FUNCTION_BLOCK GRIPPER_GIMATIC EXTENDS FB_1_Tool
VAR_INPUT
	    
    pUR : POINTER TO ROBOT_UR; // UR instance that physically carries this gripper.
    nToolOutput : USINT := 0; // Tool output used by the Gimatic interface.
    bGripLevel : BOOL := TRUE; // Electrical level that means "grip".
END_VAR
VAR_OUTPUT
    bConfigured : BOOL;
    bGripCmd     : BOOL;
END_VAR

VAR
    _nConfigState : USINT := 0;
END_VAR

METHOD Grip : eResult
VAR_INPUT
END_VAR
IF bGripLevel THEN
	Grip := SetGripperOutput(TRUE);
ELSE
	Grip := SetGripperOutput(FALSE);
END_IF
END_METHOD

METHOD PROTECTED onActivate : eResult
VAR_INPUT
END_VAR

VAR
	eParentResult: eResult;
	myResult: ERESULT;
END_VAR

VAR //YOUR CODE
	succ : BOOL;
END_VAR
eParentResult := SUPER^.onActivate();
myResult := NONE;

IF (pUR = 0) OR NOT bConfigured THEN
    Messenger.AddWarn(eMessageCategories.StateMachine, Path,
        'Gimatic gripper cannot activate because it is not configured');
    myResult := FAILURE;
ELSE
    myResult := SUCCESS;
END_IF

onActivate := CombineResults(eParentResult, myResult);
END_METHOD

METHOD PROTECTED onCleanup : eResult
VAR_INPUT
END_VAR

VAR
	eParentResult: eResult;
	myResult: ERESULT;
END_VAR

VAR //YOUR CODE
	succ : BOOL;
END_VAR
eParentResult := SUPER^.onCleanup();
bConfigured := FALSE;
bGripCmd := FALSE;
_nConfigState := 0;
myResult := SUCCESS;
onCleanup := CombineResults(eParentResult, myResult);
END_METHOD

METHOD PROTECTED onConfigure : eResult
VAR_INPUT
END_VAR

VAR
	eParentResult: eResult;
	myResult: ERESULT;
END_VAR

VAR //YOUR CODE
	succ : BOOL;
END_VAR
eParentResult := SUPER^.onConfigure();

//--------------------------------------------------
myResult := NONE;
//--------------------------------------------------

IF pUR = 0 THEN

    SetRecoveryMode(Mode := eRecoveryMode.ManualActionRequired);
    Messenger.AddError(
        eMessageCategories.Undefined,
        Name,
        'Gimatic gripper: pUR is not assigned'
    );

    bConfigured := FALSE;
    _nConfigState := 0;
    myResult := ERROR;

ELSIF nToolOutput > 1 THEN

    SetRecoveryMode(Mode := eRecoveryMode.ManualActionRequired);
    Messenger.AddError(
        eMessageCategories.Undefined,
        Name,
        'Gimatic gripper: nToolOutput must be 0 or 1'
    );

    bConfigured := FALSE;
    _nConfigState := 0;
    myResult := ERROR;

ELSIF pUR^.UR_COMM.Script.bError THEN

    SetRecoveryMode(Mode := eRecoveryMode.Automatic);
    Messenger.AddError(
        eMessageCategories.HardwareFailure,
        Name,
        'Gimatic gripper: URScript interface error'
    );

    bConfigured := FALSE;
    _nConfigState := 0;
    myResult := ERROR;

ELSE

    CASE _nConfigState OF

        0:
            bConfigured := FALSE;

            // Wait until URScript interface is available.
            IF pUR^.UR_COMM.Script.bOperational THEN

                succ :=
                    pUR^.UR_COMM.Script.ClearScript()
                    AND pUR^.UR_COMM.Script.AppendLine(
                        sLine := 'def plc_gripper_config():'
                    )
                    AND pUR^.UR_COMM.Script.AppendLine(
                        sLine := '  set_tool_voltage(24)'
                    );

                IF succ THEN

                    IF nToolOutput = 0 THEN

                        succ :=
                            pUR^.UR_COMM.Script.AppendLine(
                                sLine := '  set_tool_digital_output_mode(0,1)'
                            );

                    ELSE

                        succ :=
                            pUR^.UR_COMM.Script.AppendLine(
                                sLine := '  set_tool_digital_output_mode(1,1)'
                            );

                    END_IF

                END_IF

                succ := succ
                    AND pUR^.UR_COMM.Script.AppendLine(
                        sLine := 'end'
                    )
                    AND pUR^.UR_COMM.Script.SendBuffered();

                IF succ THEN
                    _nConfigState := 10;
                END_IF

            END_IF


        10:
            // Wait until the script FB starts sending.
            IF pUR^.UR_COMM.Script.bScriptSent THEN

                bConfigured := TRUE;
                _nConfigState := 100;

            ELSIF pUR^.UR_COMM.Script.bBusy THEN

                _nConfigState := 20;

            END_IF


        20:
            // Wait until sending is finished.
            IF pUR^.UR_COMM.Script.bError THEN
                SetRecoveryMode(Mode := eRecoveryMode.Automatic);
                Messenger.AddError(eMessageCategories.HardwareFailure, Name,
                    'Gimatic gripper: URScript interface error');

                _nConfigState := 0;
                bConfigured := FALSE;
                myResult := ERROR;

            ELSIF
                pUR^.UR_COMM.Script.bScriptSent
                OR NOT pUR^.UR_COMM.Script.bBusy
            THEN

                bConfigured := TRUE;
                _nConfigState := 100;

            END_IF


        100:
            bConfigured := TRUE;

            myResult := SUCCESS;

    END_CASE

END_IF

//--------------------------------------------------

onConfigure := CombineResults(
    eParentResult,
    myResult
);
END_METHOD

METHOD PROTECTED onDeactivate : eResult
VAR_INPUT
END_VAR

VAR
	eParentResult: eResult;
	myResult: ERESULT;
END_VAR

VAR //YOUR CODE
	succ : BOOL;
END_VAR
eParentResult := SUPER^.onDeactivate();
//--------------------------------------------------
myResult:=NONE;
// ----- YOUR CODE HERE (incl. Alarms) -------------

myResult:=SUCCESS;

// ----- END YOUR CODE -----------------------------
//--------------------------------------------------
onDeactivate := CombineResults(eParentResult,myResult);
END_METHOD

METHOD PROTECTED onError : eResult
VAR_INPUT
END_VAR

VAR
	eParentResult: eResult;
	myResult: ERESULT;
END_VAR

VAR //YOUR CODE
	succ : BOOL;
END_VAR
eParentResult := SUPER^.onError();
myResult := NONE;

bConfigured := FALSE;
_nConfigState := 0;

IF (pUR = 0) OR (nToolOutput > 1) THEN
    SetRecoveryMode(Mode := eRecoveryMode.ManualActionRequired);
    RequireNewAcknowledgement();
ELSIF pUR^.UR_COMM.State = eState.ErrorProcessing THEN
    SetRecoveryMode(Mode := pUR^.UR_COMM.RecoveryMode);
ELSIF pUR^.UR_COMM.Script.bBusy OR pUR^.UR_COMM.Script.bError THEN
    myResult := NONE;
ELSE
    myResult := SUCCESS;
END_IF

onError := CombineResults(eParentResult, myResult);
END_METHOD

METHOD PROTECTED onShutdown : eResult
VAR_INPUT
END_VAR

VAR
	eParentResult: eResult;
	myResult: ERESULT;
END_VAR

VAR //YOUR CODE
	succ : BOOL;
END_VAR
eParentResult := SUPER^.onShutdown();
//--------------------------------------------------
myResult:=NONE;
// ----- YOUR CODE HERE (incl. Alarms) -------------

// Do not release automatically on shutdown.
bConfigured := FALSE;
_nConfigState := 0;

myResult:=SUCCESS;


// ----- END YOUR CODE -----------------------------
//--------------------------------------------------
onShutdown := CombineResults(eParentResult,myResult);
END_METHOD

METHOD Release : eResult
VAR_INPUT
END_VAR
IF bGripLevel THEN
	Release := SetGripperOutput(FALSE);
ELSE
	Release := SetGripperOutput(TRUE);
END_IF
END_METHOD

METHOD SetGripperOutput : eResult
VAR_INPUT
	bValue: BOOL;
END_VAR
VAR
    succ : BOOL;
END_VAR

SetGripperOutput := NONE;

IF pUR = 0 THEN
    SetRecoveryMode(Mode := eRecoveryMode.ManualActionRequired);
    SetGripperOutput := ERROR;
	Messenger.AddError(eMessageCategories.MissingData,Path,'pUR is 0');
    RETURN;
END_IF

IF NOT bConfigured THEN
    SetRecoveryMode(Mode := eRecoveryMode.AcknowledgeRequired);
    SetGripperOutput := ERROR;
	Messenger.AddError(eMessageCategories.StateMachine,Path,'Gripper is not configured: OnConfigure');
    RETURN;
END_IF

IF pUR^.UR_COMM.Script.bError THEN
    SetRecoveryMode(Mode := eRecoveryMode.AcknowledgeRequired);
    SetGripperOutput := ERROR;
	Messenger.AddError(eMessageCategories.Undefined,Path,'UR_COMM is in Error');
    RETURN;
END_IF

// Do not overwrite a URScript command that is already being transmitted.
IF pUR^.UR_COMM.Script.bBusy THEN
    RETURN;
END_IF

IF NOT pUR^.UR_COMM.Script.ClearScript() THEN
    RETURN;
END_IF

IF NOT pUR^.UR_COMM.Script.AppendLine(
    sLine := 'def plc_grip():'
) THEN
    SetGripperOutput := ERROR;
    RETURN;
END_IF

IF nToolOutput = 0 THEN

    IF bValue THEN
        succ := pUR^.UR_COMM.Script.AppendLine(
            sLine := '  set_tool_digital_out(0,True)'
        );
    ELSE
        succ := pUR^.UR_COMM.Script.AppendLine(
            sLine := '  set_tool_digital_out(0,False)'
        );
    END_IF

ELSIF nToolOutput = 1 THEN

    IF bValue THEN
        succ := pUR^.UR_COMM.Script.AppendLine(
            sLine := '  set_tool_digital_out(1,True)'
        );
    ELSE
        succ := pUR^.UR_COMM.Script.AppendLine(
            sLine := '  set_tool_digital_out(1,False)'
        );
    END_IF

ELSE
    SetRecoveryMode(Mode := eRecoveryMode.ManualActionRequired);
    SetGripperOutput := ERROR;
    Messenger.AddError(eMessageCategories.StateMachine, Path, 'Invalid Gimatic tool output');
    RETURN;
END_IF

succ := succ
    AND pUR^.UR_COMM.Script.AppendLine(
        sLine := 'end'
    )
    AND pUR^.UR_COMM.Script.SendBuffered();

IF succ THEN
    bGripCmd := TRUE;
    SetGripperOutput := SUCCESS;
ELSE
    SetRecoveryMode(Mode := eRecoveryMode.AcknowledgeRequired);
    SetGripperOutput := ERROR;
    Messenger.AddError(eMessageCategories.HardwareFailure, Path,
        'Gimatic command send failed; physical gripper state is unknown');
END_IF
END_METHOD

END_FUNCTION_BLOCK

(* stored: Version 1.1.0.1, ProductVersion 3.1.4026.18
   POU GRIPPER_GIMATIC: Id {befc1911-49ee-4aa2-9869-a561c1fc2106}, SpecialFunc None
   Folder StateControl: Id {523b0350-c1ac-489e-b1b9-8e56cf3492cc}
   Method Grip: Id {299eaac2-c77e-45ca-9d5b-726f9f712b2e}
   Method onActivate: Id {92f80a54-c2e8-4ef0-8099-da80346a4861}
   Method onCleanup: Id {54299e02-9203-4a72-ad75-ec243ec029a6}
   Method onConfigure: Id {e3c6eab6-7f06-41e4-9710-2d10778b37ca}
   Method onDeactivate: Id {84bd92e9-04cb-4af4-bda6-a1092828e72a}
   Method onError: Id {9e9e8299-356c-4f00-8b8b-69a7f98e5a3a}
   Method onShutdown: Id {72ae2591-2fbb-4176-82c0-98cf4de0cac0}
   Method Release: Id {c9ffbe63-9dac-4121-909c-f842eb850f45}
   Method SetGripperOutput: Id {2bf51a20-cf39-4143-8eaa-eeb8a51db0c5} *)
